FUNCTION_BLOCK FB_Furnace
VAR_INPUT
END_VAR
VAR_OUTPUT
	bSaltCoverOn				   : BOOL;	
	aiSaltTemp				AT %I* : USINT;
END_VAR

END_FUNCTION_BLOCK

(* stored: Version 1.1.0.1, ProductVersion 3.1.4024.9
   POU FB_Furnace: Id {33587298-d4a9-409c-8fb0-adcf99367898}, SpecialFunc None *)
